(* PLC project cmd_motor_1d1s, Dassault Systèmes ControlBuild 2024x *)
(* stored: creationDateTime 2023-10-03T11:13:34-01:00 *)

FUNCTION_BLOCK actuator
  VAR_INPUT
    autoMode : BOOL := false;
    manualMode : BOOL := false;
  END_VAR
  VAR_INPUT
    autoCmd : BOOL := false;
  END_VAR
  VAR_INPUT
    forwardPB : BOOL := false;
    stopPB : BOOL := false;
  END_VAR
  VAR_INPUT
    generalFault : BOOL := false;
  END_VAR
  VAR_OUTPUT
    forwardCmd : BOOL := false;
  END_VAR

(* LD diagram, written out as Structured Text *)
1:
forwardCmd := (autoMode AND autoCmd OR manualMode AND (forwardPB OR forwardCmd) AND NOT stopPB) AND NOT generalFault;
END_FUNCTION_BLOCK

FUNCTION_BLOCK faults
  VAR_INPUT
    forwardCmd : BOOL := false;
  END_VAR
  VAR_INPUT
    thermalFB : BOOL := false;
    forwardFB : BOOL := false;
  END_VAR
  VAR_INPUT
    acknowledgePB : BOOL := false;
  END_VAR
  VAR_OUTPUT
    generalFault : BOOL := false;
  END_VAR
  VAR
    thermalFault : BOOL := false;
    forwardFault : BOOL := false;
  END_VAR

(* LD diagram, written out as Structured Text *)
1:
IF acknowledgePB THEN thermalFault := FALSE; END_IF;
IF acknowledgePB THEN forwardFault := FALSE; END_IF;
IF acknowledgePB THEN generalFault := FALSE; END_IF;
2:
TON_FB(IN := forwardCmd, PT := T#0h0m2s0ms);
IF TON_FB.Q0 AND NOT forwardFB THEN forwardFault := TRUE; END_IF;
3:
IF NOT thermalFB THEN thermalFault := TRUE; END_IF;
4:
IF forwardFault OR thermalFault THEN generalFault := TRUE; END_IF;
END_FUNCTION_BLOCK

(* Command of a motor with one direction and one speed and with fault detection *)
PROGRAM cmd_equipment_library.cmd_motor_1d1s
  VAR_INPUT
    autoMode : BOOL := false;
    manualMode : BOOL := false;
  END_VAR
  VAR_INPUT
    autoCmd : BOOL := false;
  END_VAR
  VAR_INPUT
    forwardFB : BOOL := false;
    thermalFB : BOOL := false;
  END_VAR
  VAR_INPUT
    forwardPB : BOOL := false;
    stopPB : BOOL := false;
  END_VAR
  VAR_INPUT
    acknowledgePB : BOOL := false;
  END_VAR
  VAR_OUTPUT
    forwardCmd : BOOL := false;
  END_VAR
  VAR_OUTPUT
    generalFault : BOOL := false;
  END_VAR

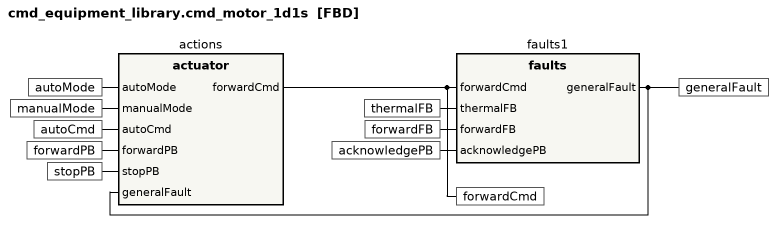
(* FBD diagram, written out as Structured Text *)
faults1(forwardCmd := actions.forwardCmd, thermalFB := thermalFB, forwardFB := forwardFB, acknowledgePB := acknowledgePB);
actions(autoMode := autoMode, manualMode := manualMode, autoCmd := autoCmd, forwardPB := forwardPB, stopPB := stopPB, generalFault := faults1.generalFault);
forwardCmd := actions.forwardCmd;
generalFault := faults1.generalFault;
END_PROGRAM
